TYPE stDIGInputsDevice :
STRUCT
	{attribute addProperty Name "Common Fault"}
	CommonFault : BIT;
	{attribute addProperty Name "Overtemperature Device"}
	OvertemperatureDevice: BIT;
	{attribute addProperty Name "Undervoltage"}
	Undervoltage : BIT;
	{attribute addProperty Name "Missing Voltage"}
	MissingVoltage : BIT;
END_STRUCT
END_TYPE

(* stored: Version 1.1.0.1, ProductVersion 3.1.4024.9
   DUT stDIGInputsDevice: Id {4dcfea83-177a-0673-17ed-cc9201a4dd6f} *)
